// TIA Portal V16 export
// export: Created 2022-07-21T09:35:25.062762Z, ExportSetting WithDefaults, DisplayName Totally Integrated Automation Portal, DisplayVersion V16 Update 4, DisplayName TIA Portal Version Control Interface, DisplayVersion V16 Update 2, DisplayName TIA Portal Openness, DisplayVersion V16 Update 4, DisplayName SINAMICS Startdrive Advanced, DisplayVersion V16 Update 5, DisplayName SINAMICS Startdrive G130, G150, S120, S150, SINAMICS MV, S210, DisplayVersion V16 Update 5, DisplayName SINAMICS Startdrive G110M, G120, G120C, G120D, G120P, G115D, DisplayVersion V16 Update 5, DisplayName STEP 7 Professional, DisplayVersion V16 Update 4, DisplayName STEP 7 Safety, DisplayVersion V16, DisplayName WinCC Advanced, DisplayVersion V16 Update 4
FUNCTION_BLOCK "fbSPEntryLReal"   // FB902, LAD
TITLE = Entry Real value / Zapis wartości Real
{ S7_Optimized_Access := 'TRUE' }
AUTHOR : a32thzz
VERSION : 0.1
// stored: AutoNumber false, IsIECCheckEnabled false, IsRetainMemResEnabled false, MemoryReserve 100, SetENOAutomatically false, UDAEnableTagReadback false
   VAR_INPUT
      max : LReal;
      min : LReal;
   END_VAR
   VAR_OUTPUT
      setpointActual : LReal;
      setpointChange : Bool;
      setpointBad : Bool;
   END_VAR
   VAR_IN_OUT
      setpointEntered : LReal;
   END_VAR
   VAR
      instTmrSetpointBad : IEC_TIMER;
      instTmrSetpointChange : IEC_TIMER;
   END_VAR
   VAR_TEMP
      setpointOK : Bool;
   END_VAR
   VAR_TEMP   // added for the SCL form of the ladder/FBD networks
      _w1 : Bool;
   END_VAR
BEGIN

REGION Network 1: Check if value is in range / Sprawdzenie czy wartość mieści się w zakresie
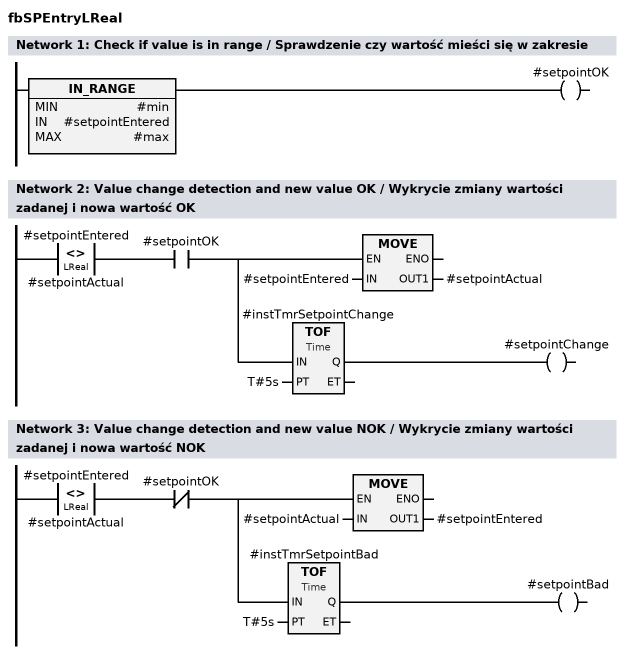
   RUNG wire#powerrail
      { S7_Templates := "SrcType := LReal" } InRange(min := #min, in := #setpointEntered, max := #max)
      Coil( #setpointOK )
   END_RUNG
   // the same network as SCL:
   #setpointOK := (#min <= #setpointEntered) AND (#setpointEntered <= #max);
END_REGION

REGION Network 2: Value change detection and new value OK / Wykrycie zmiany wartości zadanej i nowa wartość OK
   RUNG wire#powerrail
      { S7_Templates := "SrcType := LReal" } NE_Contact(in1 := #setpointEntered, in2 := #setpointActual)
      Contact( #setpointOK )
      wire#w1
      Move(in := #setpointEntered, out1 => #setpointActual)
   END_RUNG
   RUNG wire#w1
      { S7_Templates := "time_type := Time" } #instTmrSetpointChange.TOF(pt := T#5s, et =>)
      Coil( #setpointChange )
   END_RUNG
   // the same network as SCL:
   #_w1 := (#setpointEntered <> #setpointActual) AND #setpointOK;
   IF #_w1 THEN #setpointActual := #setpointEntered; END_IF;
   #instTmrSetpointChange.TOF(IN := #_w1, PT := T#5s);
   #setpointChange := #instTmrSetpointChange.Q;
END_REGION

REGION Network 3: Value change detection and new value NOK / Wykrycie zmiany wartości zadanej i nowa wartość NOK
   RUNG wire#powerrail
      { S7_Templates := "SrcType := LReal" } NE_Contact(in1 := #setpointEntered, in2 := #setpointActual)
      I_Contact( #setpointOK )
      wire#w1
      Move(in := #setpointActual, out1 => #setpointEntered)
   END_RUNG
   RUNG wire#w1
      { S7_Templates := "time_type := Time" } #instTmrSetpointBad.TOF(pt := T#5s, et =>)
      Coil( #setpointBad )
   END_RUNG
   // the same network as SCL:
   #_w1 := (#setpointEntered <> #setpointActual) AND NOT #setpointOK;
   IF #_w1 THEN #setpointEntered := #setpointActual; END_IF;
   #instTmrSetpointBad.TOF(IN := #_w1, PT := T#5s);
   #setpointBad := #instTmrSetpointBad.Q;
END_REGION
END_FUNCTION_BLOCK
